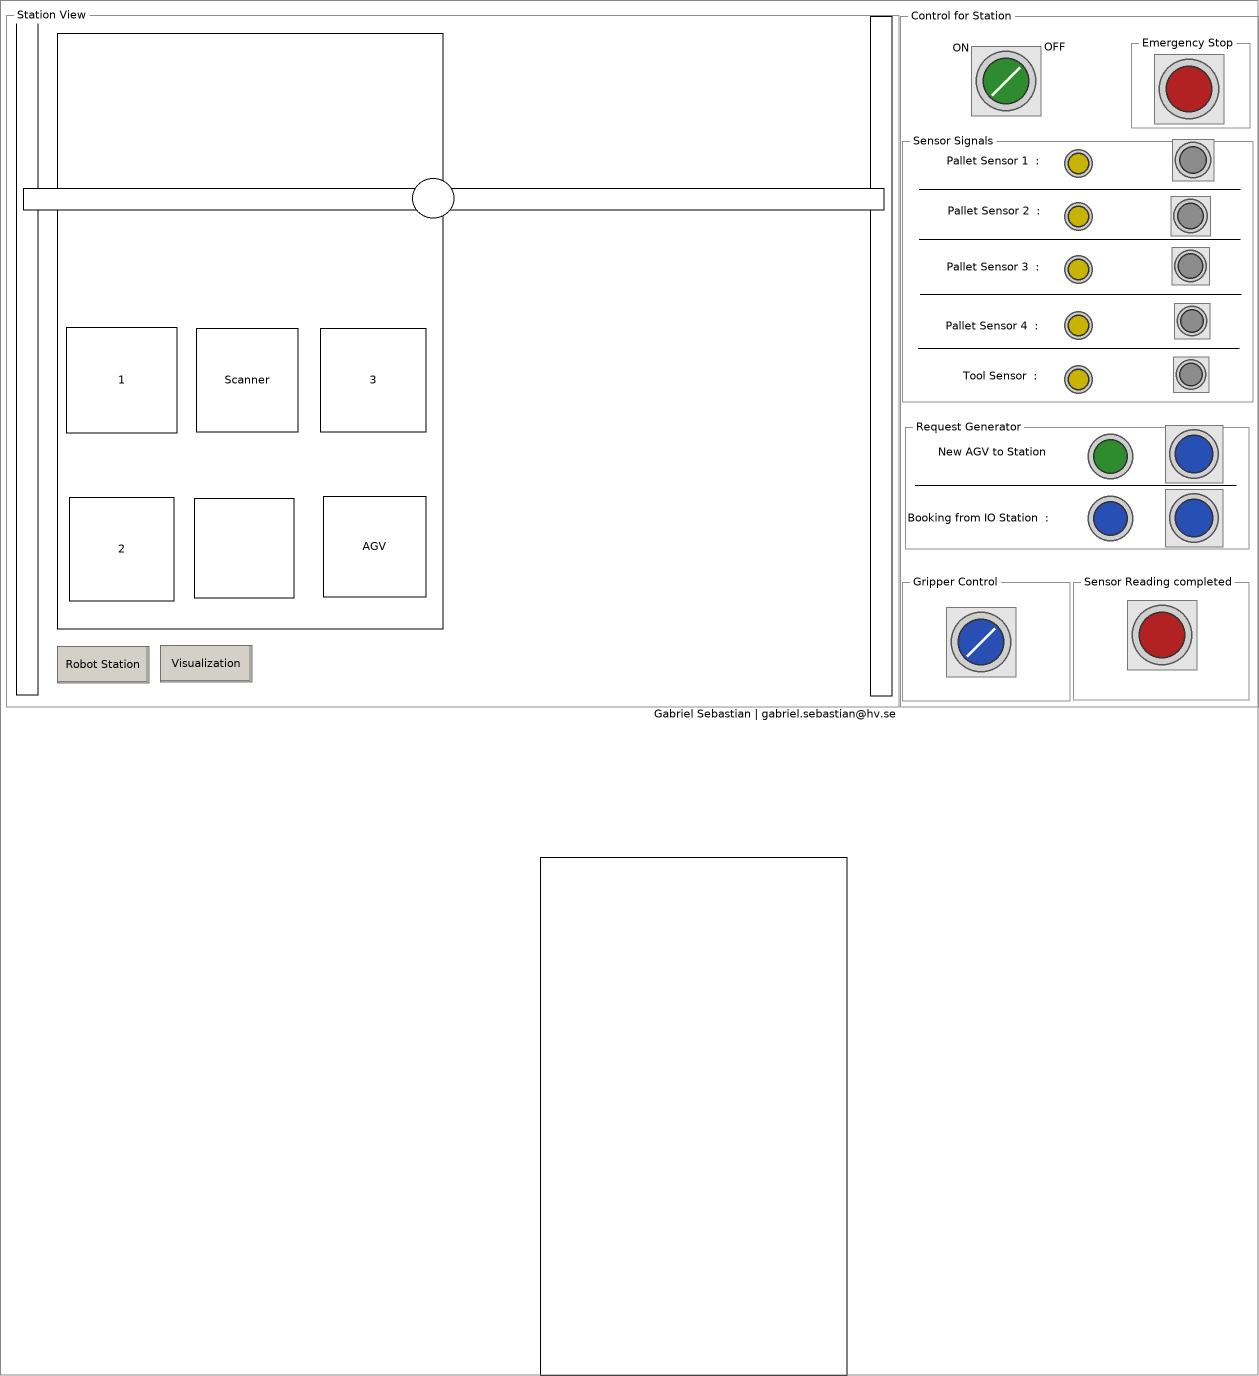
VISUALIZATION Station  // 1259x1376
    RoundedRectangle (540,857 307x519)
        p2738717112: CommData.mwCurrentAGVPOS
    Rectangle (16,15 22x680)
    GroupBox (6,7 893x700), "Station View"
        Rectangle (51,26 386x596)
        Rectangle (864,9 22x680)
        Rectangle (188,491 100x100)
        Rectangle (317,489 103x101), "AGV"
        Rectangle (190,321 102x104), "Scanner"
        Rectangle (60,320 111x106), "1"
        Rectangle (314,321 106x104), "3"
        Rectangle (63,490 105x104), "2"
        RoundedRectangle (17,181 861x22)
            p2738717112: CommData.mwYaxis
        Ellipse (406,171 42x40)
            p2738717112: CommData.mwYaxis
            p3560616238: CommData.mwXaxis
        Button (154,638 92x37), "Visualization"
            OnMouseClick: change screen: Visualization
        Button (51,639 92x37), "Robot Station"
            OnMouseClick: change screen: RobotStation
    GroupBox (900,8 359x699), "Control for Station"
        GroupBox (2,125 351x269), "Sensor Signals"
            Label (15,178 150x30), "Pallet Sensor 4 :"
            Label (17,63 150x30), "Pallet Sensor 2 :"
            Label (16,13 150x30), "Pallet Sensor 1 :"
            Line (17,56) (338,56)
            Lamp1 (160,14 33x33), variable: GVL.ixInductiveSensor1, style: Lamp-Lamp1-Yellow
            Lamp1 (160,67 33x33), variable: GVL.ixInductiveSensor2, style: Lamp-Lamp1-Yellow
            Lamp1 (160,120 33x33), variable: GVL.ixInductiveSensor3, style: Lamp-Lamp1-Yellow
            Lamp1 (160,176 33x33), variable: GVL.ixInductiveSensor4, style: Lamp-Lamp1-Yellow
            Label (16,119 150x30), "Pallet Sensor 3 :"
            Label (23,228 150x30), "Tool Sensor :"
            Lamp1 (160,230 33x33), variable: GVL.ixInductiveSensorinTool, style: Lamp-Lamp1-Yellow
            PushSwitch (266,6 50x42), variable: GVL.ixInductiveSensor1, input disabled if: CommData.mxRobotOnline, behaviour: TOGGLE, style: Switch-PushSwitch-Gray
            PushSwitch (267,63 43x40), variable: GVL.ixInductiveSensor2, input disabled if: CommData.mxRobotOnline, behaviour: TOGGLE, style: Switch-PushSwitch-Gray
            PushSwitch (269,114 39x38), variable: GVL.ixInductiveSensor3, input disabled if: CommData.mxRobotOnline, behaviour: TOGGLE, style: Switch-PushSwitch-Gray
            PushSwitch (270,170 40x36), variable: GVL.ixInductiveSensor4, input disabled if: CommData.mxRobotOnline, behaviour: TOGGLE, style: Switch-PushSwitch-Gray
            PushSwitch (271,223 36x37), variable: GVL.ixInductiveSensorinTool, input disabled if: CommData.mxRobotOnline, behaviour: TOGGLE, style: Switch-PushSwitch-Gray
            Line (17,106) (338,106)
            Line (18,161) (339,161)
            Line (16,215) (337,215)
        RotarySwitch (71,38 70x70), variable: CommData.mxOnlineMode, invisible if: CommData.mxRobotOnline, behaviour: TOGGLE, style: Switch-RotarySwitch-Green
        Label (106,24 98x30), "OFF", invisible if: CommData.mxRobotOnline
        Label (12,25 98x30), "ON", invisible if: CommData.mxRobotOnline
        GroupBox (5,411 344x130), "Request Generator"
            Label (12,18 150x30), "New AGV to Station"
            Line (10,66) (331,66)
            Lamp1 (177,11 57x53), variable: GVL.ixAGVatStation, style: Lamp-Lamp1-Green
            Lamp1 (177,73 57x53), variable: CommData.mxNewBookingrequest, style: Lamp-Lamp1-Blue
            PushSwitch (259,70 60x58), variable: CommData.mxNewBookingrequest, behaviour: TOGGLE, style: Switch-PushSwitch-Blue
        GroupBox (173,566 176x126), "Sensor Reading completed", invisible if: NOT CommData.mxWaitingforSensorinput
            PushSwitch (54,26 70x70), variable: CommData.mxScannernoobject, behaviour: TAP, style: Switch-PushSwitch-Red
        GroupBox (2,566 168x127), "Gripper Control"
            Lamp1 (-1748,-553 70x70), style: Lamp-Lamp1-Yellow
            Lamp1 (44,34 70x70), variable: CommData.mxGripper, style: Lamp-Lamp1-Yellow
            RotarySwitch (44,33 70x70), variable: CommData.mxGripper, invisible if: NOT Visualaisation_Control.mxManualMode, behaviour: TOGGLE, style: Switch-RotarySwitch-Blue
        GroupBox (231,27 119x93), "Emergency Stop"
            PushSwitch (23,19 70x70), variable: GVL.ixEmergencyStop, behaviour: TOGGLE, style: Switch-PushSwitch-Red
    Label (900,503 156x30), "Booking from IO Station :"
    Label (650,699 250x30), "Gabriel Sebastian | gabriel.sebastian@hv.se"
    PushSwitch (1164,425 60x58), variable: CommData.mxRequestAGV, behaviour: TOGGLE, style: Switch-PushSwitch-Blue
END_VISUALIZATION

(* stored: Version 1.1.0.1, ProductVersion 3.1.4024.12
   Visu Station: Id {890bd767-353b-46f4-949f-665e4f3e5b85} *)
